TYPE ConveyorOutput :
STRUCT
	SensorDataOutput : ARRAY[0..10] OF SensorOutput;
	SensorNum : DINT;
	//Ramps
	RampDataOutput : ARRAY[0..5] OF SensorOutput;
	RampNum : DINT;
	//Pushers
	PusherOut : ARRAY[0..10] OF SensorOutput;
	PusherNum : DINT;
	//Motor Output
	MotorOutput : MotorOutput;
END_STRUCT
END_TYPE

(* stored: Version 1.1.0.1
   DUT ConveyorOutput: Id {cfade488-78f4-49a6-8a42-5629f32f8a73} *)
